TYPE ST_StorageSlot :
STRUCT
	nStorageId : INT;
	nStorageName : STRING;
	bMaintanence : BOOL;
END_STRUCT
END_TYPE

(* stored: Version 1.1.0.1, ProductVersion 3.1.4024.16
   DUT ST_StorageSlot: Id {b4bdd010-1420-44b8-bbb5-775ccb5e0217} *)
